INTERFACE I_TrafficLight

METHOD M_Beep : BOOL
VAR_INPUT
	/// On/Off signal
	bEnable:				BOOL;
	/// Flashing frequency (0 = Permanently On, 1 = 1s alternately, ...)
	uiBlinkFrequency:		UINT;
END_VAR
END_METHOD

METHOD M_Green : BOOL
VAR_INPUT
	/// On/Off light
	bEnable:				BOOL;
	/// Flashing frequency (0 = Permanently On, 1 = 1s alternately, ...)
	uiBlinkFrequency:		UINT;
	/// Reset all colors, before set this color
	bResetOther:			BOOL;
END_VAR
END_METHOD

METHOD M_Multicolor : BOOL
VAR_INPUT
	/// Enable green
	bGreen:					BOOL;
	/// Enable yellow
	bYellow:				BOOL;
	/// Enable red
	bRed:					BOOL;
	/// Flashing frequency (0 = Permanently On, 1 = 1s alternately, ...)
	uiBlinkFrequency:		UINT;
END_VAR
END_METHOD

METHOD M_Red : BOOL
VAR_INPUT
	/// On/Off light
	bEnable:				BOOL;
	/// Flashing frequency (0 = Permanently On, 1 = 1s alternately, ...)
	uiBlinkFrequency:		UINT;
	/// Reset all colors, before set this color
	bResetOther:			BOOL;
END_VAR
END_METHOD

METHOD M_Reset : BOOL
VAR_INPUT
END_VAR
END_METHOD

METHOD M_Yellow : BOOL
VAR_INPUT
	/// On/Off light
	bEnable:				BOOL;
	/// Flashing frequency (0 = Permanently On, 1 = 1s alternately, ...)
	uiBlinkFrequency:		UINT;
	/// Reset all colors, before set this color
	bResetOther:			BOOL;
END_VAR
END_METHOD

PROPERTY P_BeepState : BOOL
GET
END_GET
END_PROPERTY

PROPERTY P_GreenState : BOOL
GET
END_GET
END_PROPERTY

PROPERTY P_RedState : BOOL
GET
END_GET
END_PROPERTY

PROPERTY P_YellowState : BOOL
GET
END_GET
END_PROPERTY

END_INTERFACE

(* stored: Version 1.1.0.1, ProductVersion 3.1.4024.12
   Itf I_TrafficLight: Id {23cd0bc1-e28e-4991-afd7-9230b5c9a16d}
   Method M_Beep: Id {bb056172-509c-4431-b8f0-d3b84e61d9d9}
   Method M_Green: Id {5392e748-f362-4b4e-b841-c08a07fab4c7}
   Method M_Multicolor: Id {3b6fcb6b-4cdb-40a3-8698-c2b5ff82a1be}
   Method M_Red: Id {9d04d6c2-6410-4453-8b7a-cf3835f0ce9e}
   Method M_Reset: Id {05f4770d-7654-4978-9007-3f4a01dd27bf}
   Method M_Yellow: Id {290ab3ce-12ac-4bb0-ae6c-1cc3e1a605b5}
   Property P_BeepState: Id {79a2d464-12eb-48cd-941e-7595f1af30f9}
   Get Get: Id {057a686d-e852-4bb3-8651-6ebebe48fa63}
   Property P_GreenState: Id {231624c7-da4a-47de-9e17-56cdadcfaaab}
   Get Get: Id {44d0d2d1-e807-49cc-80a7-f0928ebd0860}
   Property P_RedState: Id {36aa8f5c-94f0-40ba-a92b-4d9d66f51e9d}
   Get Get: Id {04da49f1-a004-4f79-89b4-47e5ce8eecea}
   Property P_YellowState: Id {f77d27da-9cf1-44db-b33f-c9db4bc66884}
   Get Get: Id {03bc0115-a94a-4d76-8d32-8e78a04f21fc} *)
